PROGRAM MAIN
VAR
	fbStateMachine : FB_StateMachine;
END_VAR


fbStateMachine();

END_PROGRAM

(* stored: Version 1.1.0.1, ProductVersion 3.1.4024.11
   POU MAIN: Id {5538f496-a75c-45f1-9bad-d338e8535694}, SpecialFunc None *)
